TYPE "FeedMachine_Wng"
VERSION : 0.1
// Block: FeedMachine_Wng
   STRUCT
      NotAutReady : Bool;
      MissingCnd_Bkw : Bool;
      MissingCnd_Fwd : Bool;
      Ax : TAx_Warnings;
   END_STRUCT;

END_TYPE
